// TIA Portal project "Buffer Station" (V17)

(* hardware
DEVICE "S71500/ET200MP-Station_1"  S7-1500 station
   slot 0: "Profilschiene_0"  6ES7 590-1***0-0AA0
   slot 1: "PLC_1"  CPU 1511-1 PN  6ES7 511-1AK00-0AB0  V1.8
   slot 2: "AI 8xU/I/RTD/TC ST_1"  AI 8xU/I/RTD/TC ST  6ES7 531-7KF00-0AB0  V2.0
   slot 3: "AI 8xU/I/RTD/TC ST_2"  AI 8xU/I/RTD/TC ST  6ES7 531-7KF00-0AB0  V2.0
   slot 4: "AI 8xU/I/RTD/TC ST_3"  AI 8xU/I/RTD/TC ST  6ES7 531-7KF00-0AB0  V2.0
   slot 5: "AI 8xU/I/RTD/TC ST_4"  AI 8xU/I/RTD/TC ST  6ES7 531-7KF00-0AB0  V2.0
   slot 6: "DI 16x24VDC BA_1"  DI 16x24VDC BA  6ES7 521-1BH10-0AA0  V1.0
*)

// ===== PLC "PLC_1"  CPU 1511-1 PN =====

VAR_GLOBAL   // PLC tag table "Standard-Variablentabelle"
   "AT BUFFER ENTRY" AT %E0.0 : Bool;
   "AT BUFFER EXİT" AT %I0.1 : Bool;
   "AT EXİT" AT %I0.2 : Bool;
   "START" AT %I0.3 : Bool;
   "RESET" AT %I0.4 : Bool;
   "STOP" AT %I0.5 : Bool;
   "AUTO" AT %I0.6 : Bool;
   "EMERGENCY STOP" AT %I0.7 : Bool;
   "BUFFER VEL." AT %ID30 : Real;
   "STOP BLADE" AT %Q0.0 : Bool;
   "START LİGHT" AT %Q0.1 : Bool;
   "RESET LİGHT" AT %Q0.2 : Bool;
   "STOP LİGHT" AT %Q0.3 : Bool;
   "BUFFER CONVEYOR" AT %QD30 : Real;
   "EXİT CONVEYOR" AT %QD34 : Real;
   "COUNTER" AT %QD38 : DInt;
   "Tag_1" AT %M0.0 : Bool;
   "Tag_2" AT %MD100 : DWord;
   "Tag_3" AT %MD200 : DWord;
   "Tag_4" AT %M0.1 : Bool;
   "Tag_5" AT %M0.2 : Bool;
   "Tag_6" AT %M0.4 : Bool;
   "Tag_7" AT %M0.3 : Bool;
   "Tag_8" AT %M0.6 : Bool;
   "Tag_9" AT %MW100 : Int;
END_VAR

// folder: System blocks/Program resources

DATA_BLOCK "IEC_Counter_0_DB"   // DB1
{ S7_Optimized_Access := 'TRUE' }
AUTHOR : Simatic
FAMILY : IEC
NAME : CNTR
VERSION : 1.0
// stored: InstanceOfName IEC_COUNTER
"IEC_COUNTER"
BEGIN
END_DATA_BLOCK

// folder: (top level)

FUNCTION "MHJ-PLC-Lab-Function-S71500" : Void   // FC9000, SCL
{ S7_Optimized_Access := 'TRUE' }
VERSION : 0.1
   VAR_TEMP
      Value : Byte;
      ForCounter : Int;
   END_VAR
   VAR CONSTANT
      Value_01_DW : DWord := 16#1223_5486;
      Value_02_DW : DWord := 16#A6C9_D1F5;
   END_VAR
BEGIN

   #Value:=PEEK(area := 16#82,
        dbNumber := 0,
        byteOffset := 511);
   #Value := #Value + 1;

   POKE(area := 16#82,
        dbNumber := 0,
        byteOffset := 511,
        value := #Value);

   POKE(area := 16#82,
        dbNumber := 0,
        byteOffset := 1016,
        value := #Value_01_DW);
   POKE(area := 16#82,
        dbNumber := 0,
        byteOffset := 1020,
        value := #Value_02_DW);

   FOR #ForCounter := 0 TO 63 DO
       #Value:=PEEK(area := 16#1,
            dbNumber := 0,
            byteOffset := #ForCounter);
       POKE(area := 16#81,
            dbNumber := 0,
            byteOffset := #ForCounter,
            value := #Value);
   END_FOR;
   #Value := PEEK(area := 16#1,
                  dbNumber := 0,
                  byteOffset := 512);
   POKE(area := 16#82,
        dbNumber := 0,
        byteOffset := 512,
        value := #Value);
END_FUNCTION

ORGANIZATION_BLOCK "Main"   // OB1, LAD, ProgramCycle
TITLE = "Main Program Sweep (Cycle)"
{ S7_Optimized_Access := 'TRUE' }
VERSION : 0.1
   VAR_INPUT
      Initial_Call : Bool;   // Initial call of this OB
      Remanence : Bool;   // =True, if remanent data are available
   END_VAR
   VAR_TEMP   // added for the SCL form of the ladder/FBD networks
      _w1 : Bool;
      _w2 : Bool;
   END_VAR
BEGIN

REGION Network 1
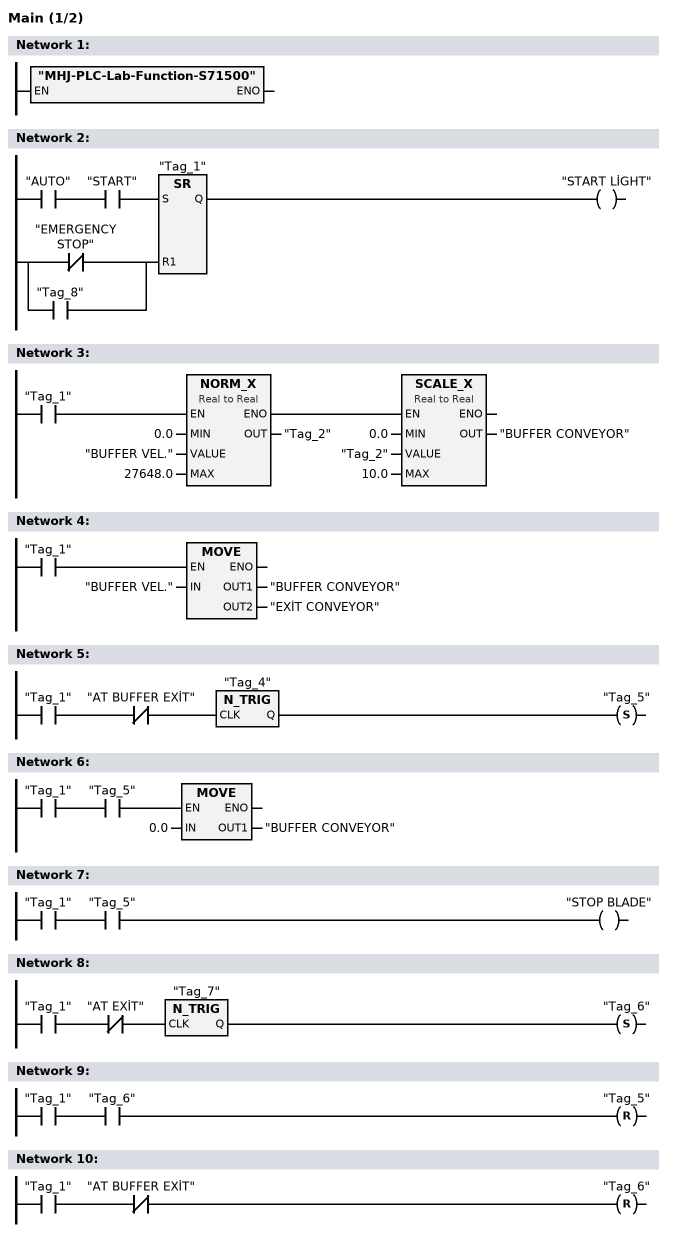
   RUNG wire#powerrail
      "MHJ-PLC-Lab-Function-S71500"()
   END_RUNG
   // the same network as SCL:
   "MHJ-PLC-Lab-Function-S71500"();
END_REGION

REGION Network 2
   RUNG wire#powerrail
      Contact( "AUTO" )
      Contact( "START" )
      S_SR(operand := "Tag_1", r1 := wire#w1)
      Coil( "START LİGHT" )
   END_RUNG
   RUNG wire#powerrail
      I_Contact( "EMERGENCY STOP" )
   END_RUNG wire#w1
   RUNG wire#powerrail
      Contact( "Tag_8" )
   END_RUNG wire#w1
   // the same network as SCL:
   IF "AUTO" AND "START" THEN
       "Tag_1" := TRUE;   // SR flip-flop
   END_IF;
   IF NOT "EMERGENCY STOP" OR "Tag_8" THEN "Tag_1" := FALSE; END_IF;
   "START LİGHT" := "Tag_1";
END_REGION

REGION Network 3
   RUNG wire#powerrail
      Contact( "Tag_1" )
      { S7_Templates := "[SrcType := Real, DestType := Real]" } Normalize(min := 0.0, value := "BUFFER VEL.", max := 27648.0, out => "Tag_2")
      { S7_Templates := "[SrcType := Real, DestType := Real]" } Scale(min := 0.0, value := "Tag_2", max := 10.0, out => "BUFFER CONVEYOR")
   END_RUNG
   // the same network as SCL:
   IF "Tag_1" THEN
       "Tag_2" := NORM_X(MIN := 0.0, VALUE := "BUFFER VEL.", MAX := 27648.0);
       "BUFFER CONVEYOR" := SCALE_X(MIN := 0.0, VALUE := "Tag_2", MAX := 10.0);
   END_IF;
END_REGION

REGION Network 4
   RUNG wire#powerrail
      Contact( "Tag_1" )
      Move(in := "BUFFER VEL.", out1 => "BUFFER CONVEYOR", out2 => "EXİT CONVEYOR")
   END_RUNG
   // the same network as SCL:
   IF "Tag_1" THEN
       "BUFFER CONVEYOR" := "BUFFER VEL.";
       "EXİT CONVEYOR" := "BUFFER VEL.";
   END_IF;
END_REGION

REGION Network 5
   RUNG wire#powerrail
      Contact( "Tag_1" )
      I_Contact( "AT BUFFER EXİT" )
      N_Trig( "Tag_4" )
      S_Coil( "Tag_5" )
   END_RUNG
   // the same network as SCL:
   #_w1 := "Tag_1" AND NOT "AT BUFFER EXİT";
   #_w2 := NOT #_w1 AND "Tag_4";   // falling edge
   "Tag_4" := #_w1;
   IF #_w2 THEN "Tag_5" := TRUE; END_IF;
END_REGION

REGION Network 6
   RUNG wire#powerrail
      Contact( "Tag_1" )
      Contact( "Tag_5" )
      Move(in := 0.0, out1 => "BUFFER CONVEYOR")
   END_RUNG
   // the same network as SCL:
   IF "Tag_1" AND "Tag_5" THEN "BUFFER CONVEYOR" := 0.0; END_IF;
END_REGION

REGION Network 7
   RUNG wire#powerrail
      Contact( "Tag_1" )
      Contact( "Tag_5" )
      Coil( "STOP BLADE" )
   END_RUNG
   // the same network as SCL:
   "STOP BLADE" := "Tag_1" AND "Tag_5";
END_REGION

REGION Network 8
   RUNG wire#powerrail
      Contact( "Tag_1" )
      I_Contact( "AT EXİT" )
      N_Trig( "Tag_7" )
      S_Coil( "Tag_6" )
   END_RUNG
   // the same network as SCL:
   #_w1 := "Tag_1" AND NOT "AT EXİT";
   #_w2 := NOT #_w1 AND "Tag_7";   // falling edge
   "Tag_7" := #_w1;
   IF #_w2 THEN "Tag_6" := TRUE; END_IF;
END_REGION

REGION Network 9
   RUNG wire#powerrail
      Contact( "Tag_1" )
      Contact( "Tag_6" )
      R_Coil( "Tag_5" )
   END_RUNG
   // the same network as SCL:
   IF "Tag_1" AND "Tag_6" THEN "Tag_5" := FALSE; END_IF;
END_REGION

REGION Network 10
   RUNG wire#powerrail
      Contact( "Tag_1" )
      I_Contact( "AT BUFFER EXİT" )
      R_Coil( "Tag_6" )
   END_RUNG
   // the same network as SCL:
   IF "Tag_1" AND NOT "AT BUFFER EXİT" THEN "Tag_6" := FALSE; END_IF;
END_REGION

REGION Network 11
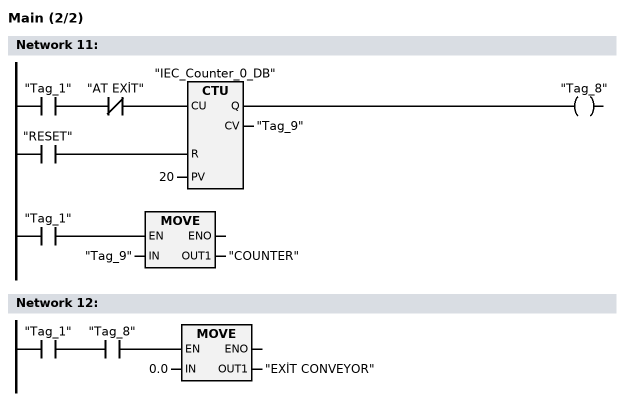
   "IEC_Counter_0_DB".CTU(CU := "Tag_1" AND NOT "AT EXİT", R := "RESET", PV := 20, CV => "Tag_9");
   "Tag_8" := "IEC_Counter_0_DB".Q;
   IF "Tag_1" THEN "COUNTER" := "Tag_9"; END_IF;
END_REGION

REGION Network 12
   RUNG wire#powerrail
      Contact( "Tag_1" )
      Contact( "Tag_8" )
      Move(in := 0.0, out1 => "EXİT CONVEYOR")
   END_RUNG
   // the same network as SCL:
   IF "Tag_1" AND "Tag_8" THEN "EXİT CONVEYOR" := 0.0; END_IF;
END_REGION
END_ORGANIZATION_BLOCK